(* IEC 61131-3 sources: SRCI/RobotLibrary/Library/POUs/General/MC_CreateServerLog_ToDo, 1 file *)

(* ---- MC_CreateServerLog_ToDo.st ---- *)
FUNCTION_BLOCK MC_CreateServerLog_ToDo EXTENDS RobotLibraryBaseFB
VAR
END_VAR

END_FUNCTION_BLOCK

METHOD FB_init : BOOL
VAR_INPUT
  /// if TRUE, the retain variables are initialized (warm start / cold start)
  bInitRetains : BOOL;
  /// if TRUE, the instance afterwards gets moved into the copy code (online change)
  bInCopyCode  : BOOL;
END_VAR

  MyType := 'MC_CreateServerLogFB';

  ExecMode := ExecutionMode.PARALLEL;
  Priority := PriorityLevel.NORMAL;

END_METHOD
